(* CODESYS project MIC7001_fulldemo.2020.1218.1.project

Project tree, tasks and I/O mapping:
  Device : Changsha-Cyber-MI-linux, Changsha Cyber-MI Co., Ltd., version 3.5.10.40
    application Application
      libraries: Standard, * (System); SysFile, 3.5.15.0 (System); SysTypes2 Interfaces, * (System); SysShm, * (System); CAA Mathematics, * (CAA Technical Workgroup); SysTime, 3.5.9.0 (System); CAA Types Extern, 3.5.13.0 (CAA Technical Workgroup); CAA DTUtil Extern, 3.5.12.0 (CAA Technical Workgroup); Util, * (System); TCP, 3.5.15.0 (3S - Smart Software Solutions GmbH); CAA Net Base Services, 3.5.15.0 (CAA Technical Workgroup); MIC7001 base library, 0.99 (Cyber-MI.com); CAA SerialCom, 3.5.15.0 (CAA Technical Workgroup); CAN API, 1.0.0.3 (3S - Smart Software Solutions GmbH)
      task task_slow (cyclic, interval 200 ms, priority 30, watchdog 900 ms x 10) calls prg_retain, prg_set_inmode
      task task_middle (cyclic, interval 100 ms, priority 20, watchdog 500 ms x 5) calls prg_mqtt, prg_data2file, prg_can0_cfc, prg_485
      task task_fast (cyclic, interval 20 ms, priority 10, watchdog 300 ms x 10) calls prg_init, prg_input, prg_main, prg_can1_st, prg_output
      Enums/
        data type pi_index
      programs/
        program prg_set_inmode [CFC]
        program prg_init [ST]
        program prg_mqtt [CFC]: find_key, ACT_first_buffer, ACT_running_light, proc_set_command, ACT_boot, ACT_normal_buffer, ACT_publish, proc_get_command, ACT_recv_proc
        program prg_data2file [ST]
        program prg_retain [ST]
        program prg_can0_cfc [CFC]: recv_301, send_f007
        program prg_can1_st [ST]
        program prg_input [ST]
        program prg_output [ST]
        program prg_main [ST]
        program prg_485 [ST]
      global variables GVL
      trace Trace (task task_fast): prg_main.AI_01, prg_main.AI_02
      global variables PersistentVars
    IoDrvMIC7001 : IoDrvMIC7001, Cyber-MI, version 19.1.1
        input  Application.prg_main.AI_01 : DWORD  // Ai55_Pwm-i2
        input  Application.prg_main.AI_02 : DWORD  // Ai56_Pwm-i3
        output Application.prg_output.ao_00 : DWORD  // Ao00-Ai46@C22
        output Application.prg_output.ao_01 : DWORD  // Ao01-Ai47@D14
        output Application.prg_output.led_run : BOOL  // LED_run
        output Application.prg_output.led_err : BOOL  // LED_err
        output Application.prg_output.led_usr : BOOL  // LED_usr
        unmapped channels: Ai00@C16, Ai01@C28, Ai02@C17, Ai03@C29, Ai04@C30, Ai05@C19, Ai06@C31, Ai07@C20, Ai08@C18, Ai09@D18, Ai10@D20, Ai11@D31, Ai12@D19, Ai13@D30, Ai14@D29, Ai15@D17, Ai16@D28, Ai17@D16, Ai18-Do00@C25, Ai19-Do01@C24, Ai20-Do02@C13, Ai21-Do03@C01, Ai22-Do04@C03, Ai23-Do05@C04, Ai24-Do06@C05, Ai25-Do07@C06, Ai26-Do08@C08, Ai27-Do09@C09, Ai28-Do10@C10, Ai29-Do11@C11, Ai30-Do12@D34, Ai31-Do13@D35, Ai32-Do14@D23, Ai33-Do15@D12, Ai34-Do16@D10, Ai35-Do17@D09, Ai36-Do18@D08, Ai37-Do19@D07, Ai38-Do20@D05, Ai39-Do21@D04,
          Ai40-Do22@D03, Ai41-Do23@D02, Ai42-Do24@C23, Ai43-Do25@C35, Ai44-Do26@D24, Ai45-Do27@D13, Ai46-Ao00@C22, Ai47-Ao01@D14, Ai48_Pi02, Ai49_Out5V, Ai50_VCC, Ai51_VCC_L, Ai52_VCC_R, Ai53_Pwm-i0, Ai54_Pwm-i1, Ai57_CPU-T, Ai58_G-x, Ai59_G-y, Ai60_G-z, Ai61-reserved, Ai62-IO-cntr, Ai63-CDS-cntr, Di00-Ai00@C16, Di01-Ai01@C28, Di02-Ai02@C17, Di03-Ai03@C29, Di04-Ai04@C30, Di05-Ai05@C19, Di06-Ai06@C31, Di07-Ai07@C20, Di08-Ai08@C18, Di09-Ai09@D18, Di10-Ai10@D20, Di11-Ai11@D31, Di12-Ai12@D19, Di13-Ai13@D30, Di14-Ai14@D29, Di15-Ai15@D17, Di16-Ai16@D28, Di17-Ai17@D16,
          Di18-Ai18@C25, Di19-Ai19@C24, Di20-Ai20@C13, Di21-Ai21@C01, Di22-Ai22@C03, Di23-Ai23@C04, Di24-Ai24@C05, Di25-Ai25@C06, Di26-Ai26@C08, Di27-Ai27@C09, Di28-Ai28@C10, Di29-Ai29@C11, Di30-Ai30@D34, Di31-Ai31@D35, Di32-Ai32@D23, Di33-Ai33@D12, Di34-Ai34@D10, Di35-Ai35@D09, Di36-Ai36@D08, Di37-Ai37@D07, Di38-Ai38@D05, Di39-Ai39@D04, Di40-Ai40@D03, Di41-Ai41@D02, Di42-Ai42@C23, Di43-Ai43@C35, Di44-Ai44@D24, Di45-Ai45@D13, Di46-Ai46@C22, Di47-Ai47@D14, Di48-Pi00@C15, Di49-Pi01@C14, Di50-Pi02@D22, Di51-Pi03@D21, Di52-reserved, Di53-reserved, Di54-reserved, Di55-reserved, Di56-reserved, Di57-reserved,
          Di58-reserved, Di59-reserved, Di60-reserved, Di61-reserved, Di62-reserved, Di63-reserved, Pi00-Di48@C15, Pi01-Di49@C14, Pi02-Di50@D22, Pi03-Di51@D21, Do00-Ai18@C25, Do01-Ai19@C24, Do02-Ai20@C13, Do03-Ai21@C01, Do04-Ai22@C03, Do05-Ai23@C04, Do06-Ai24@C05, Do07-Ai25@C06, Do08-Ai26@C08, Do09-Ai27@C09, Do10-Ai28@C10, Do11-Ai29@C11, Do12-Ai30@D34, Do13-Ai31@D35, Do14-Ai32@D23, Do15-Ai33@D12, Do16-Ai34@D10, Do17-Ai35@D09, Do18-Ai36@D08, Do19-Ai37@D07, Do20-Ai38@D05, Do21-Ai39@D04, Do22-Ai40@D03, Do23-Ai41@D02, Do24-Ai42@C23, Do25-Ai43@C35, Do26-Ai44@D24, Do27-Ai45@D13, Do28-Pwmi00@C33, Do29-Pwmi01@C34,
          Do30-Pwmi02@D25, Do31-Pwmi03@D26, PWM00@C25, PWM01@C24, PWM02@C13, PWM03@C01, PWM04@C03, PWM05@C04, PWM06@C05, PWM07@C06, PWM08@C08, PWM09@C09, PWM10@C10, PWM11@C11, PWM12@D34, PWM13@D35, PWM14@D23, PWM15@D12, PWM16@D10, PWM17@D09, PWM18@D08, PWM19@D07, PWM20@D05, PWM21@D04, PWM22@D03, PWM23@D02, PWM24@C23, PWM25@C35, PWM26@D24, PWM27@D13, PWM28-Pwmi00@C33, PWM29-Pwmi01@C34, PWM30-Pwmi02@D25, PWM31-Pwmi03@D26, PWM_I_0@C33, PWM_I_1@C34, PWM_I_2@D25, PWM_I_3@D26, ctrl_ai_raw, ctrl_adjust,
          ctrl_adj0, ctrl_adj1, ctrl_adj2, ctrl_adj3, disable_5V
    SoftMotion General Axis Pool
  libraries: VisuSymbols, 3.5.10.0 (System)
  5ce3da45-db07-42e7-a21c-a00fff4ed8f6|C:\Users\zhou\p01.bmp
  5ce3da45-db07-42e7-a21c-a00fff4ed8f6|C:\working\p01.bmp
  5ce3da45-db07-42e7-a21c-a00fff4ed8f6|C:\working\file.bmp
  text list GlobalTextList
*)

// Device/Application/Enums/pi_index
(*掉电保持参数定义*)
TYPE pi_index :
(
	current_01_max := 0,  // 电磁阀1最大电流， 第一个需要赋值为0， 后面的不需赋值，会自动累加
	current_01_min,       // 电磁阀1最小电流
	current_02_max,
	current_02_min,
	current_03_max,
	current_03_min         // 最后一个不用逗号
	
	// 可在这里添加需要保存的参数, 最多255个
	
);
END_TYPE

// Device/Application/GVL
{attribute 'qualified_only'}
VAR_GLOBAL
	// MIC7001 基本信息，从控制器内部读取
	mysn:STRING(32);  // MIC7001 序列号 类似： CMI010320090123
	iccid:STRING(32); // MIC7001 内部sim卡序列号
	lac:STRING(8);    // GSM 小区号
	cid:STRING(8);    // GSM 基站号
	r_mins:DINT;  // 运行时间 分钟数
	
	//retain 变量, 建议放在全局变量列表 gvl中
	g_retain01:ARRAY[0..mic7001_base.Constants.RETAIN_NUM_MAX] OF DINT;	
	g_retain_ok:BOOL := FALSE;  // retain变量正常标志, 为 true 则说明retain变量可用
	
	// 模拟量输出设定值
	ao_00_in:DWORD := 0;  // 模拟量输出通道 00   单位： mV
	ao_01_in:DWORD := 0;  // 模拟量输出通道 01   单位： mV
	
	
END_VAR

// Device/Application/PersistentVars
{attribute 'qualified_only'}
VAR_GLOBAL PERSISTENT RETAIN
	myRetain01:DWORD;
END_VAR

// Device/Application/programs/prg_retain
PROGRAM prg_retain
VAR
	inited:BOOL := FALSE;
	
	// 每组retain变量可以保存100个参数，如果不够，可创建第二个
	// 下面的change.me.txt.01 这个名字最好修改成其它的，避免跟其它机型重复，造成售后万一调换控制器后参数混淆
	myRetain01:mic7001_base.FB_RETAIN := (filename := '/userdata/change.me.txt.01', use_bak := TRUE);  
	
	// 如果上面的100个参数不够用，可以打开下面这两行的注释 ，增加另外100个
(*	myRetain02:mic7001_base.FB_RETAIN := (filename := '/userdata/retain.txt.02', use_bak := TRUE);
	g_retain02:ARRAY[0..mic7001_base.Constants.RETAIN_NUM_MAX] OF DINT;	
*)	
END_VAR

//步骤一：初始化默认值,如果读取文件失败，则使用默认值作为当前参数
IF NOT inited THEN  //上电执行一次，设置retain变量的缺省值
	//第一组retain变量初始值，新控制器第一次上电有效。
	myRetain01.default_val[pi_index.current_01_max] := 800;
	myRetain01.default_val[pi_index.current_01_min] := 200;
	myRetain01.default_val[pi_index.current_02_max] := 800;
	myRetain01.default_val[pi_index.current_02_min] := 200;
	myRetain01.default_val[pi_index.current_03_max] := 800;
	myRetain01.default_val[pi_index.current_03_min] := 200;
	
	//第二组retain变量初始值，新控制器第一次上电有效。
(*	myRetain02.default_val[0] := 999;
	myRetain02.default_val[1] := 888;
	myRetain02.default_val[2] := 777;
	// .....
	myRetain02.default_val[98] := 333;
	myRetain02.default_val[99] := 222;  //最后一个
*)	
	inited := TRUE;
END_IF

//步骤二：执行功能块，处理参数的保存和读取
myRetain01(value := gvl.g_retain01);
gvl.g_retain_ok := myRetain01.ok;

(*
myRetain02(value := g_retain02);
*)

//步骤三：在其它任务中直接使用 gvl.g_retain01[] 作为retain变量

END_PROGRAM

// Device/Application/programs/prg_set_inmode
PROGRAM prg_set_inmode
VAR
	FB_SET_INMODE_0: MIC7001_BASE.FB_SET_INMODE;
END_VAR

VAR CONSTANT
	MODE_5V: 	UINT := 0;
	MODE_36V:	UINT := 1;
	MODE_20mA:	UINT := 2;
	MODE_30K : 	UINT := 3;
	MODE_DI_H: 	UINT := 4;
	MODE_DI_L: 	UINT := 5;
END_VAR

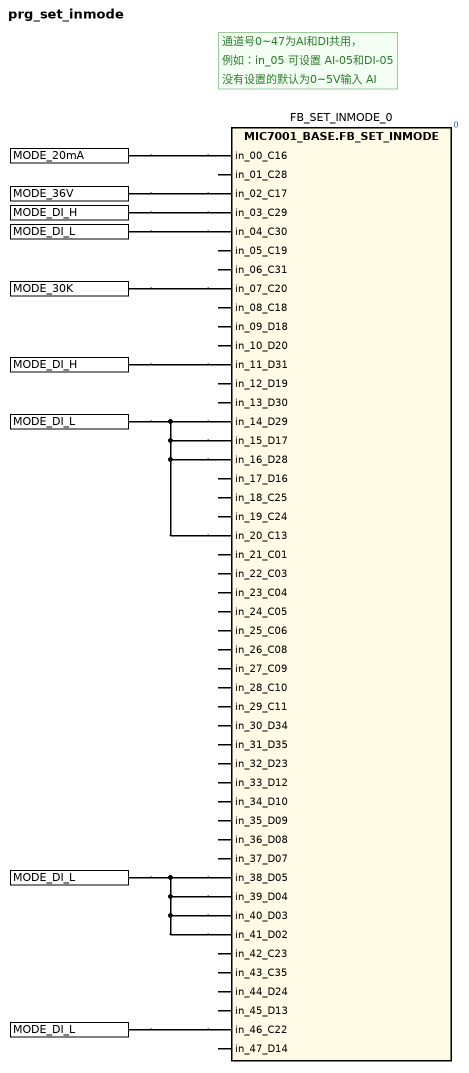
// 通道号0~47为AI和DI共用，
// 例如：in_05 可设置 AI-05和DI-05
// 没有设置的默认为0~5V输入 AI
FB_SET_INMODE_0(
    in_00_C16 := MODE_20mA,
    in_02_C17 := MODE_36V,
    in_03_C29 := MODE_DI_H,
    in_04_C30 := MODE_DI_L,
    in_07_C20 := MODE_30K,
    in_11_D31 := MODE_DI_H,
    in_14_D29 := MODE_DI_L,
    in_15_D17 := MODE_DI_L,
    in_16_D28 := MODE_DI_L,
    in_20_C13 := MODE_DI_L,
    in_38_D05 := MODE_DI_L,
    in_39_D04 := MODE_DI_L,
    in_40_D03 := MODE_DI_L,
    in_41_D02 := MODE_DI_L,
    in_46_C22 := MODE_DI_L); // MIC7001_BASE.FB_SET_INMODE

END_PROGRAM

// Device/Application/programs/prg_mqtt
PROGRAM prg_mqtt
VAR
	FB_MQTTClient_0: mic7001_base.FB_MQTTClient;
	payload : STRING(255) := '{"RPM": 1234, "Hours": 2345}';
	xPub : BOOL := FALSE;
	xSub : BOOL := FALSE;
	xBooted :BOOL := FALSE;
	
	ton_pub : ton; 
	
	val_payload:ARRAY[0..32] OF mic7001_base.dut_json;
	rpm_value : DINT := 1000;
	hours_value :REAL := 680;
	time_value : STRING;
	sn_value : STRING(128);
	lac_str:STRING(128);
	cid_str:STRING(128);
	press_value :REAL := 20.1;
	
	recv_data : ARRAY[0..32] OF mic7001_base.DUT_json;
	old_recv_cntr:UDINT := 0;
	payload_len :INT;
	
	mqtt_first :BOOL := TRUE;
	ton_running:ton:=(pt := T#500MS);
	pkg_id :DINT := 0;
	i :DINT;
	hour_today:REAL := 2.0;
	
	xLock_cmd : BOOL := FALSE;
	diLock_grade : DINT := 0;
	diLock_delay : DINT := 0;
	mqtt_interval : DINT := 5;  //mqtt package interval of publish to server	
	cntr_wait_sub : INT := 0;
END_VAR

VAR CONSTANT
	TYPE_DINT:UINT := 0;
	TYPE_REAL:UINT := 1;
	TYPE_STRING:UINT := 2;
END_VAR

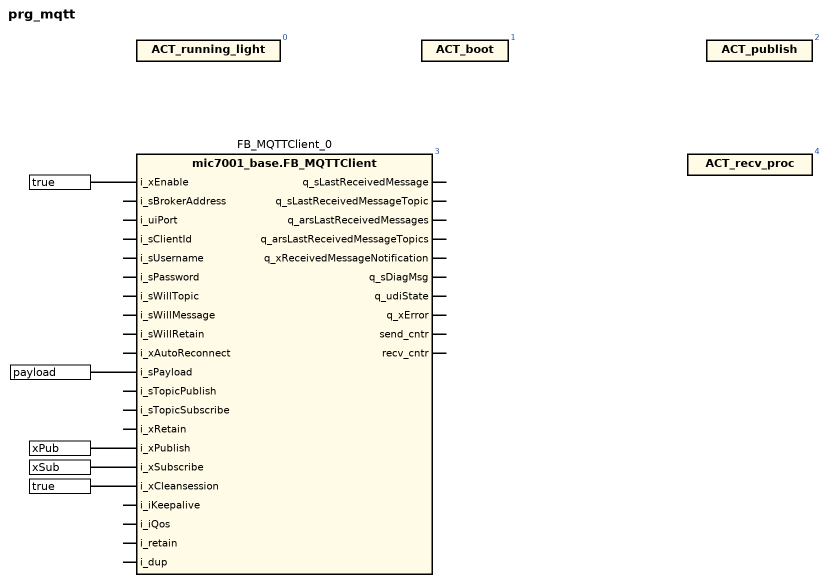
ACT_running_light();
ACT_boot();
ACT_publish();
FB_MQTTClient_0(
    i_xEnable := true,
    i_sPayload := payload,
    i_xPublish := xPub,
    i_xSubscribe := xSub,
    i_xCleansession := true); // mic7001_base.FB_MQTTClient
ACT_recv_proc();

METHOD find_key : dint
VAR_INPUT
	key :STRING(32);
END_VAR
VAR
	i :UINT;
END_VAR
find_key := -1;

FOR i := 0 TO payload_len-1 DO
	IF key = recv_data[i].key THEN
		find_key := i;
		RETURN;
	END_IF
END_FOR

RETURN; // not find,  return -1
END_METHOD

ACTION ACT_first_buffer:

val_payload[0].key := 'sn';
val_payload[0].val_tp := TYPE_STRING;
IF MIC7001_base.read_sn(ADR(sn_value)) THEN
	val_payload[0].value_str := sn_value;
ELSE
	val_payload[0].value_str := 'SN Error';
END_IF

val_payload[1].key := 'lac';
val_payload[1].val_tp := TYPE_STRING;

val_payload[2].key := 'cid';
val_payload[2].val_tp := TYPE_STRING;

IF MIC7001_base.read_location(lac := ADR(lac_str), ci := ADR(cid_str)) THEN
	val_payload[1].value_str := lac_str; 
	val_payload[2].value_str := cid_str; 
ELSE
	val_payload[1].value_str := 'lac_error'; 
	val_payload[2].value_str := 'cid_error'; 
END_IF

val_payload[3].key := 'work_mins';
val_payload[3].val_tp := TYPE_DINT;
val_payload[3].value_dint := MIC7001_base.read_work_mins();

payload := mic7001_base.arr2json(arr := val_payload, num := 4);
END_ACTION

ACTION ACT_running_light:
ton_running(in := NOT ton_running.Q);
IF ton_running.Q THEN
	prg_output.led_usr := FALSE;
END_IF

IF FB_MQTTClient_0.q_udiState <> 60 THEN
	prg_output.led_usr := TRUE;
END_IF
END_ACTION

ACTION proc_set_command:
(*
	cmd:  	set  	          	//命令字, set:设置参数或者执行命令，  get：点播数据或参数
	interval:	15				//设置上传间隔： 15秒
	act:  	lock, unlock		//锁机动作类型
	grade:  1, 2, 3, 4			//动作级别
	delay:  0, 60, 3600			//延迟时间,单位： 秒
*)

// check lock command 
i := find_key(key := 'act');
IF i >= 0 AND recv_data[i].val_tp = mic7001_base.Constants.TYPE_STRING  THEN
	IF recv_data[i].value_str = 'lock' THEN
		xlock_cmd := TRUE;
	ELSIF recv_data[i].value_str = 'unlock' THEN
		xlock_cmd := FALSE;
	END_IF
END_IF

i := find_key(key := 'grade');
IF i >= 0 AND recv_data[i].val_tp = mic7001_base.Constants.TYPE_DINT THEN
	diLock_grade := recv_data[i].value_dint;
END_IF

i := find_key(key := 'delay');
IF i >= 0 AND recv_data[i].val_tp = mic7001_base.Constants.TYPE_DINT THEN
	diLock_delay := recv_data[i].value_dint;
END_IF

i := find_key(key := 'interval');
IF i >= 0 AND recv_data[i].val_tp = mic7001_base.Constants.TYPE_DINT THEN
	mqtt_interval := recv_data[i].value_dint;
END_IF
END_ACTION

ACTION ACT_boot:
IF NOT xbooted THEN
	IF FB_MQTTClient_0.q_udiState = 60 THEN
		xSub := TRUE;
		xBooted := TRUE;
	END_IF
END_IF
END_ACTION

ACTION ACT_normal_buffer:

val_payload[0].key := 'rpm';
val_payload[0].val_tp := mic7001_base.Constants.TYPE_DINT; 
rpm_value := rpm_value + 8;
IF rpm_value > 2200 THEN
	rpm_value := 1000;
END_IF
val_payload[0].value_dint := rpm_value; 

val_payload[1].key := 'hour_all';
val_payload[1].val_tp := mic7001_base.Constants.TYPE_REAL;
hours_value := hours_value +  ANY_TO_REAL(mqtt_interval)/3600;
val_payload[1].value_real := hours_value; 

val_payload[2].key := 'power';
val_payload[2].val_tp := mic7001_base.Constants.TYPE_REAL;  
val_payload[2].value_real := ANY_TO_REAL(rpm_value)/10.0 - 39.0; 

val_payload[3].key := 'press';
val_payload[3].val_tp := mic7001_base.Constants.TYPE_REAL;  
press_value := ANY_TO_REAL(rpm_value)*1.5/100;
IF press_value > 35 THEN
	press_value := 35;
ELSIF press_value < 2 THEN
	press_value := 2;
END_IF
val_payload[3].value_real := press_value; 

val_payload[4].key := 'fuel_all';
val_payload[4].val_tp := mic7001_base.Constants.TYPE_REAL;  
val_payload[4].value_real := ANY_TO_REAL(hours_value)*13.2; 

val_payload[5].key := 'fuel_rate';
val_payload[5].val_tp := mic7001_base.Constants.TYPE_REAL; 
val_payload[5].value_real := press_value/9.1; 

val_payload[6].key := 'work_all';
val_payload[6].val_tp := mic7001_base.Constants.TYPE_REAL;
val_payload[6].value_real := hours_value*97.2; 

val_payload[7].key := 'hour_today';
val_payload[7].val_tp := mic7001_base.Constants.TYPE_REAL;
hour_today := hour_today + ANY_TO_REAL(mqtt_interval)/3600;
IF hour_today > 9 THEN
	hour_today := 2.0;
END_IF
val_payload[7].value_real := hour_today; 

val_payload[8].key := 'fuel_today';
val_payload[8].val_tp := mic7001_base.Constants.TYPE_REAL;
val_payload[8].value_real := hour_today*12.3; 

val_payload[9].key := 'work_today';
val_payload[9].val_tp := mic7001_base.Constants.TYPE_REAL;
val_payload[9].value_real := hour_today*97.2; 


payload := mic7001_base.arr2json(arr := val_payload, num := 10);
END_ACTION

ACTION ACT_publish:
IF FB_MQTTClient_0.q_udiState <> 60 THEN   //not ready, return and wait
	xPub := FALSE;
	RETURN;
END_IF

cntr_wait_sub := cntr_wait_sub + 1;
IF cntr_wait_sub < 10 THEN   // wait for subscribe succeed
	RETURN;
END_IF

IF mqtt_first THEN
	mqtt_first := FALSE;
	ACT_first_buffer();
	FB_MQTTClient_0.i_register := TRUE;
	xPub := TRUE;
	RETURN;
END_IF

ton_pub(in := NOT ton_pub.Q, pt := ANY_TO_TIME(mqtt_interval*1000));   // second to ms
IF ton_pub.Q THEN
	ACT_normal_buffer();
	FB_MQTTClient_0.i_register := FALSE;
	xPub := TRUE;
ELSE
	xPub := FALSE;
END_IF
END_ACTION

ACTION proc_get_command:
(*
	cmd:  	get  	//命令字, get：点播数据或参数
	rpm:  	15		//点播转速， 上传15次
	press:  0		//点播压力， 持续上传
	fuel_all: 1	  	//点播总油耗，上传一次 					
*)
END_ACTION

ACTION ACT_recv_proc:
(*
	cmd:  	set, get          			//命令字, set:设置参数或者执行命令，  get：点播数据或参数
	act:  	lock, unlock, reboot		//动作类型
	grade:  1, 2, 3, 4					//动作级别
	delay:  0, 60, 3600					//延迟时间,单位： 秒
*)

IF old_recv_cntr = FB_MQTTClient_0.recv_cntr THEN  //no new message
	RETURN;
END_IF
old_recv_cntr := FB_MQTTClient_0.recv_cntr;

payload_len := mic7001_base.json2arr(json := FB_MQTTClient_0.q_sLastReceivedMessage, pArr := ADR(recv_data), max_len := 32);
IF payload_len = 0 THEN
	RETURN;
END_IF

i := find_key(key := 'cmd');
IF i >= 0 AND recv_data[i].val_tp = mic7001_base.Constants.TYPE_STRING THEN 
	IF  recv_data[i].value_str = 'get' THEN
		proc_get_command();
	ELSIF recv_data[i].value_str = 'set' THEN
		proc_set_command();
	END_IF
END_IF
END_ACTION

END_PROGRAM

// Device/Application/programs/prg_output
PROGRAM prg_output
VAR
	ton_run:ton;
	
	ao_00:DWORD;  // 需要绑定到AO端口表中
	ao_01:DWORD;  // 需要绑定到AO端口表中
	ao_adj:mic7001_base.FB_AO_ADJ;  
		
END_VAR

VAR_INPUT
	led_run : BOOL := TRUE;
	led_usr : BOOL := FALSE;
	led_err : BOOL := FALSE;	
END_VAR


 //运行灯 每秒闪烁一次运行灯
ton_run(in := NOT ton_run.Q, pt := T#0.5S); 
IF ton_run.Q THEN
	led_run := NOT led_run;
END_IF

// 使用 AO 端口的校准参数
ao_adj(xEnable := TRUE, in_ao_00_mv := gvl.ao_00_in, in_ao_01_mv := gvl.ao_01_in, out_ao_00 => ao_00, out_ao_01 => ao_01, xErr =>);

END_PROGRAM

// Device/Application/programs/prg_data2file
PROGRAM prg_data2file
VAR
	data:ARRAY[0..MIC7001_base.Constants.FILE_DATA_MAX] OF REAL;
	data2file :MIC7001_base.FB_DATA2FILE;
	save_data:BOOL := FALSE;
END_VAR

// 根据实际情况，判断是否需要保存数据， 如果需要，则设置save_data 为 true
data2file.xEnable := save_data;

IF save_data THEN
	data[0] := 12345;  //发动机转速
	data[1] := 33333;  //主泵压力
	data[2] := 44444;  //液压油温
	data[3] := 55555;  //油门旋钮
	data[4] := 66666;  //燃油油位
END_IF

data2file(data := data,    			// 待保存的数组 
		length := 5, 				// 数组内需要保存的数据个数
		interval := T#200MS, 		// 保存间隔， 本例中 每隔200毫秒保存一次，每次将data数组中的前个数据写入数据文件，增加一行
		filedir := '/userdata/', 	// 文件保存路径，无需更改。 本路径空间为2.6G， 保存的文件名为开始记录数据的时间，例如： /userdata/2020.1.2.15.23.45.csv
		maxsize_m := 10);			// 单个文件的大小限制（单位：兆）， 本例中，如果数据文件大小达到10Mbytes， 则自动停止记录。 
									// 等到下次 save_data由false -> true时, 会新创建一个文件，继续记录

END_PROGRAM

// Device/Application/programs/prg_can0_cfc
PROGRAM prg_can0_cfc  // CAN 功能块 CFC语言例程， 需要安装 mic7001_baselib V0.96或以上版本
VAR
	CAN0: MIC7001_BASE.FB_CAN0_B2B4; // 定义CAN0，
	
	// 注册需要接收的基本帧和扩展帧
    reg_11bit:ARRAY[0..63] OF UDINT :=     [301, 302, 303, 304, 60(0)];  // 注册四个基本帧id，最多支持64个，如果不够，请联系厂家定制
    timeout_11bit:ARRAY[0..63] OF UDINT := [200, 500, 800, 100, 60(0)]; // 设置四个基本帧的接收超时时间，单位： 毫秒
    
    reg_29bit:ARRAY[0..63] OF UDINT :=     [16#0CF00301, 16#0CF00401, 62(0)];  // 注册两个扩展帧id，最多支持64个，如果不够，请联系厂家定制
    timeout_29bit:ARRAY[0..63] OF UDINT := [200,         500,         62(0)]; // 设置两个扩展帧的接收超时时间，单位： 毫秒
    
    msgSend11bit:CAN.MESSAGE;
    msgSend29bit:CAN.MESSAGE;
    
    send_cmd:BOOL := FALSE;  // 需要发送数据

    recv_id:UDINT;
    recv_data:ARRAY[0..7] OF BYTE;
    
END_VAR

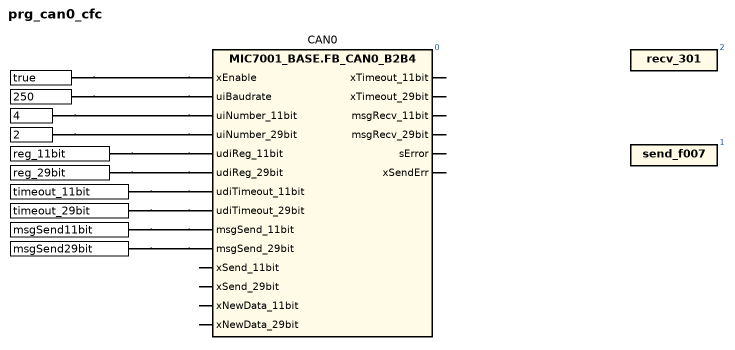
CAN0(
    xEnable := true,
    uiBaudrate := 250,
    uiNumber_11bit := 4,
    uiNumber_29bit := 2,
    udiReg_11bit := reg_11bit,
    udiReg_29bit := reg_29bit,
    udiTimeout_11bit := timeout_11bit,
    udiTimeout_29bit := timeout_29bit,
    msgSend_11bit := msgSend11bit,
    msgSend_29bit := msgSend29bit); // MIC7001_BASE.FB_CAN0_B2B4
send_f007();
recv_301();

ACTION recv_301:

IF CAN0.xNewData_11bit[0] THEN   // 收到 301 基本帧
    // 接收数据
    recv_id := CAN0.msgRecv_11bit[0].udiCanID;
    recv_data[0] := CAN0.msgRecv_11bit[0].abyData[0];
    recv_data[1] := CAN0.msgRecv_11bit[0].abyData[1];
    // ......
    recv_data[7] := CAN0.msgRecv_11bit[0].abyData[7];
    
    CAN0.xNewData_11bit[0] := FALSE;  // 清除新数据标志
	
ELSIF CAN0.xTimeout_11bit[0] THEN  // 301帧接收超时
    // 超时处理	
	
END_IF
END_ACTION

ACTION send_f007:

IF send_cmd THEN
    msgSend29bit.udiCanID := 16#0CF00701;
    msgSend29bit.usiDataLength := 8;
    msgSend29bit.abyData[0] := 1;
    msgSend29bit.abyData[1] := 1;
    msgSend29bit.abyData[2] := 23;
    msgSend29bit.abyData[3] := 21;
    msgSend29bit.abyData[4] := 12;
    msgSend29bit.abyData[5] := 45;
    msgSend29bit.abyData[6] := 56;
    msgSend29bit.abyData[7] := 78;
    CAN0.xSend_29bit := TRUE;  // 启动发送
   
    send_cmd := FALSE;
END_IF
END_ACTION

END_PROGRAM

// Device/Application/programs/prg_485
PROGRAM prg_485
VAR		
	Com1Params: 			ARRAY [1..7] OF COM.PARAMETER;	(* Settings to communicate with the COM Port *)
	hCom: 					CAA.HANDLE;
	ComOpen: 				COM.Open;
	ComClose: 				COM.Close;
	ComWrite: 				COM.Write;
	ComRead: 				COM.Read;	
	
	Snd_Cnt:				CAA.SIZE;

	Rcv_Cnt: 				CAA.SIZE;
	xCom1CloseError: 		BOOL;
	xCom1WriteError: 		BOOL;
	xCom1ReadError: 		BOOL;
	xError:					BOOL;
	
	uiComState: INT := 0;
	ComID:USINT:=8;

	cmdSend:BOOL := FALSE;
	
	Writebuffer:			ARRAY[1..16] OF BYTE;
	Readbuffer: 			ARRAY[1..16] OF BYTE;
	len_read:caa.SIZE;
	read_cntr : DINT := 0;
	send_cntr : BYTE := 0;
END_VAR

CASE uiComState OF
	0:
	Com1Params[1].udiParameterId := COM.CAA_Parameter_Constants.udiPort;
	Com1Params[1].udiValue := 8;    //MIC7001的RS485接口为串口8
	Com1Params[2].udiParameterId := COM.CAA_Parameter_Constants.udiBaudrate;
	Com1Params[2].udiValue := 115200;
	Com1Params[3].udiParameterId := COM.CAA_Parameter_Constants.udiParity;
	Com1Params[3].udiValue := INT_TO_UINT(COM.PARITY.NONE);
	Com1Params[4].udiParameterId := COM.CAA_Parameter_Constants.udiStopBits;
	Com1Params[4].udiValue := INT_TO_UINT(COM.STOPBIT.ONESTOPBIT);
	Com1Params[5].udiParameterId := COM.CAA_Parameter_Constants.udiTimeout;
	Com1Params[5].udiValue := 0;
	Com1Params[6].udiParameterId := COM.CAA_Parameter_Constants.udiByteSize;
	Com1Params[6].udiValue := 8;
	Com1Params[7].udiParameterId := COM.CAA_Parameter_Constants.udiBinary;
	Com1Params[7].udiValue := 0;					
	ComOpen(xExecute := TRUE, usiListLength:=UINT_TO_USINT(SIZEOF(Com1Params)/SIZEOF(COM.PARAMETER)),pParameterList:= ADR(Com1Params),hCom=> hCom);			
	IF ComOpen.xError THEN
		uiComState := 32767;
	ELSIF ComOpen.xDone THEN
		uiComState := 10;
	END_IF
	
	10:
		send_cntr := send_cntr +1;
		Writebuffer[5] := send_cntr;
		ComWrite(xExecute := TRUE,hCom:= hCom,pBuffer:= ADR(Writebuffer),szSize:= 5);		
		IF ComWrite.xError THEN
			uiComState := 32767;
		END_IF
		IF ComWrite.xDone THEN		
			ComRead(xExecute := FALSE);
			ComWrite(xExecute := FALSE);
			uiComState := 20;
		END_IF
	
	20:
	ComRead(xExecute := TRUE,hCom:= hCom, pBuffer:= ADR(Readbuffer), szBuffer:= SIZEOF(Readbuffer) , szsize => len_read);			
	IF ComRead.xError THEN
		uiComState := 32767;
	END_IF
	IF ComRead.xDone THEN
		ComRead(xExecute := FALSE);
		ComWrite(xExecute := FALSE);
		IF len_read = 6 THEN
			uiComState := 10;
		END_IF
	END_IF
	read_cntr := read_cntr +1;
	IF read_cntr >100 THEN
		read_cntr := 0;
		uiComState := 10;
	END_IF
	255:
	
	32767:	
END_CASE

END_PROGRAM

// Device/Application/programs/prg_init
PROGRAM prg_init
VAR
	booted :BOOL := FALSE;

	ton_mins:ton;
	
END_VAR


IF NOT booted THEN
	booted := TRUE;
	mic7001_base.set_piv01(6000);  //将 PI-00， PI-01的门槛电压设置为6V
	mic7001_base.set_piv23(8700);  //将 PI-02,  PI-03的门槛电压设置为8.7V
	
	mic7001_base.Disable_120ohm_can0();  //禁用CAN0口的内部终端电阻
	mic7001_base.Enable_120ohm_can1();  //启用CAN1口的内部终端电阻
		
	mic7001_base.read_sn(ADR(gvl.mysn));  //读取控制器序列号
	
	mic7001_base.set_pwm_frequency(0, 200);   //设置 C端口所有PWM频率为 200Hz  （范围： 50 ~  1000 Hz）
	mic7001_base.set_pwm_frequency(1, 300);   //设置 D端口所有PWM频率为 300Hz  （范围： 50 ~  1000 Hz）

	mic7001_base.read_iccid(iccid := ADR(gvl.iccid));    // 读取内部sim卡号，可作为控制器唯一标识
	mic7001_base.read_location(lac := ADR(gvl.lac), ci := ADR(gvl.cid));  //读取 GSM网络的小区号和基站号， 可通过 lbs-sir 公众号 ，输入 这两个数字查询地理位置
	gvl.r_mins := mic7001_base.read_work_mins();  // 读取控制器累计运行分钟数
END_IF

ton_mins(in := NOT ton_mins.Q, pt := T#60S);
IF ton_mins.Q THEN
	gvl.r_mins := mic7001_base.read_work_mins();  // 读取控制器累计运行分钟数
END_IF

END_PROGRAM

// Device/Application/programs/prg_input
PROGRAM prg_input
VAR
END_VAR


// 处理输入端口

END_PROGRAM

// Device/Application/programs/prg_main
PROGRAM prg_main
VAR
	AI_01:DWORD;
	AI_02:DWORD;
END_VAR

IF NOT gvl.g_retain_ok THEN   // 如果不需要retain变量， 可删除
	RETURN;
END_IF

// 主机液压系统控制

END_PROGRAM

// Device/Application/programs/prg_can1_st
PROGRAM prg_can1_st
VAR
    can1:MIC7001_BASE.FB_CAN1_A1A4;  // 定义CAN1功能块（端口号： A1--CAN_H,   A4--CAN_L）, 如果要使用CAN0， 更改为： FB_CAN0_B2B4
    inited:BOOL:= FALSE; // 初始化完成标志
    msg_recv:CAN.MESSAGE;
    id_recv:UDINT;
    timeout : BOOL ;
	send_data:ARRAY[0..7] OF BYTE;
	ton_send_801 :  ton := (pt := T#300MS);  // 801数据发送定时器
	ton_send_802 :  ton := (pt := T#500MS);  // 802数据发送定时器
	ton_send_f055 : ton := (pt := T#800MS);  // f055数据发送定时器
END_VAR


// 第一步：初始化，只需要执行一次
IF NOT inited THEN
    can1.m_set_baudrate(baudrate := 250);  // 设置波特率, 支持：  125K，250K，500K，1000K
    
    // 注册接收id
    can1.m_reg_id_11bit(id := 401, timeout := 300);  // 注册一个基本帧
    can1.m_reg_id_11bit(id := 402, timeout := 300);  // 注册一个基本帧
	// 基本帧最多注册64个， 如果不够，可联系厂家定制功能块
	
    can1.m_reg_id_29bit(id := 16#0CF00301, timeout := 300);  // 注册一个扩展帧
	can1.m_reg_id_29bit(id := 16#0CF00401, timeout := 500);  // 注册一个扩展帧
	can1.m_reg_id_29bit(id := 16#0CF00501, timeout := 100);  // 注册一个扩展帧
	can1.m_reg_id_29bit(id := 16#0CF00601, timeout := 200);  // 注册一个扩展帧
    // 扩展帧最多注册64个， 如果不够，可联系厂家定制功能块
	
    can1.m_start();  // 启动can1口，需要在注册接收id之后
    
    inited := TRUE;  // 初始化完成标志，避免再次执行
END_IF

// 第二步：执行功能块
can1();  

// 第三步：接收数据， 下面的id必须在初始化的时候进行过注册
IF can1.m_recv_msg_11bit(id := 401, pMsg := ADR(msg_recv)) > 0 THEN   //接收一个基本帧
    // 接收数据在 结构体 msg_recv 中， 根据需求进行处理
    id_recv := msg_recv.udiCanID;
    // ......
ELSIF can1.m_is_timeout_11bit(id := 401) THEN   // 没有收到数据，判断是否超时
    // 超时, 做相应处理
    timeout := TRUE;
END_IF

IF can1.m_recv_msg_29bit(id := 16#0CF00301, pMsg := ADR(msg_recv)) > 0 THEN   //接收一个扩展帧
    // 接收数据在 结构体 msg_recv 中， 根据需求进行处理
    id_recv := msg_recv.udiCanID;
    // ......
ELSIF can1.m_is_timeout_29bit(id := 16#0CF00301) THEN   // 没有收到数据，判断是否超时
    // 超时, 做相应处理
    timeout := TRUE;    
END_IF

// 第四步： 发送数据
ton_send_801(in := NOT ton_send_801.Q);
IF ton_send_801.Q THEN  // 发送 801 基本帧\
	send_data[0] := 1;
	// ......
	send_data[7] := 7;
	can1.m_send_msg_11bit(id := 801, data := send_data, len := 8);
END_IF

ton_send_802(in := NOT ton_send_802.Q);
IF ton_send_802.Q THEN  // 发送 802 基本帧\
  
	send_data[0] := 1;
	// ......
	send_data[7] := 7;
	can1.m_send_msg_11bit(id := 802, data := send_data, len := 8);
END_IF

ton_send_f055(in := NOT ton_send_f055.Q);
IF ton_send_f055.Q THEN  // 发送 f055 扩展帧
	send_data[0] := 11;
	send_data[1] := 22;
	send_data[2] := 33;
	send_data[3] := 11;
	send_data[4] := 22;
	send_data[5] := 33;
	send_data[6] := 11;
	send_data[7] := 22;
	    
	can1.m_send_msg_29bit(id := 16#01F05501, data := send_data, len := 8);
END_IF

END_PROGRAM
